(* Logix 5000 project; controller grafcet1 Emulate 5570 rev 32.11; software revision 32.00 *)

TASK MainTask (continuous, watchdog 500 ms) : MainProgram

MODULES
   Local : Emulate 5570 (ICP 2, rev 32.11)
END_MODULES

VAR_GLOBAL   (* controller tags *)
   AlarmaWrapDone : BOOL;
   Banda2ON : BOOL;
   Bandallenado : BOOL;
   BandaON : BOOL;
   BandaRechazo : BOOL;
   BandaSalida : BOOL;
   BandaTapado : BOOL;
   Cocacola6 : BOOL;
   ContadorSecuencia : DINT;
   ContadorSensorRechazo : DINT := 61;
   ContadorWrap : COUNTER := (PRE := 18, ACC := 1);
   Cortadora : BOOL;
   CrearCocacolaWrap : BOOL;
   E0 : BOOL;
   E1 : BOOL;
   E10 : BOOL;
   E11 : BOOL;
   E12 : BOOL;
   E13 : BOOL;
   E14 : BOOL;
   E15 : BOOL;
   E16 : BOOL;
   E17 : BOOL;
   E18 : BOOL;
   E19 : BOOL;
   E2 : BOOL;
   E20 : BOOL;
   E21 : BOOL;
   E22 : BOOL;
   E3 : BOOL;
   E4 : BOOL;
   E5 : BOOL;
   E6 : BOOL;
   E7 : BOOL;
   E8 : BOOL;
   E9 : BOOL;
   EliminarCocacola6 : BOOL;
   EliminarCocacolaWrap : BOOL;
   EmergencyStop : BOOL := 1;
   EN_Lineas : BOOL;
   ER2 : BOOL;
   FechaHora : DINT[7];
   GenerarCocacola6 : BOOL;
   HornoON : BOOL;
   InterceptorGiro : DINT;
   Llenador : BOOL;
   Memoria_ONS : BOOL;
   NuevaBotella : BOOL;
   NuevaBotella_Ant : BOOL;
   NumeroBotellas : COUNTER := (PRE := 1000);
   NumeroBotellasRechazadas : COUNTER := (PRE := 1000);
   NumeroLote : DINT;
   ObjetoEnHorno : BOOL;
   OffsetLote : DINT;
   ONS_Llenado : BOOL;
   ONS_SalidaTapado : BOOL;
   ONS_Secuencia : BOOL;
   PistonRechazo : BOOL;
   PorcentajeRechazo : DINT := 20;
   PosicionLote : DINT;
   PulsadorRechazo : BOOL;
   RechazoAleatorio : BOOL;
   RechazosPor10 : DINT;
   Reset : BOOL;
   Rodillos : BOOL;
   RutinaPaletizado : BOOL;
   SeisBotellasWrap : COUNTER := (PRE := 6);
   SensorCortador : BOOL;
   SensorEntraBandaSW : BOOL;
   SensorInterceptor : BOOL;
   SensorInterceptorTrabajo : BOOL;
   SensorLlenado : BOOL;
   SensorPosicionRechazo : BOOL;
   SensorPosicionRechazo_Ant : BOOL;
   SensorSaleTunelCalor : BOOL;
   SensorSalidaBandaSW : BOOL;
   SensorSalidaRechazo : BOOL;
   SensorSalidaTapado : BOOL;
   SensorTapado : BOOL;
   SensorTope : BOOL;
   SensorTunelCalor : BOOL;
   START : BOOL;
   StartCalidad : BOOL;
   StartLlenado : BOOL;
   Tapado : BOOL;
   TerminaMov : BOOL;
   TiempoWrap : TIMER := (PRE := 2000);
   Tope : BOOL;
   TuboAbajo : BOOL;
   ValorAleatorio : DINT;
END_VAR

PROGRAM MainProgram   (* main routine MainRoutine *)

ROUTINE MainRoutine   (* ladder *)
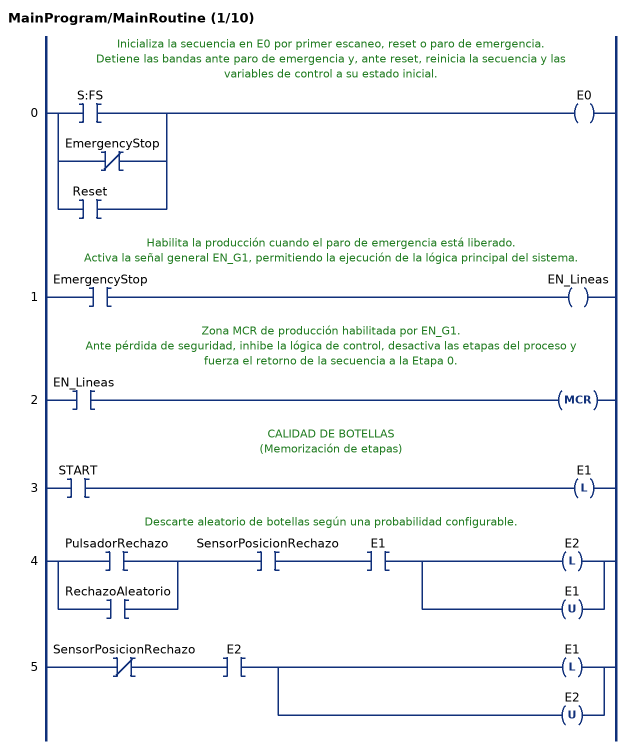
   // Inicializa la secuencia en E0 por primer escaneo, reset o paro de emergencia.
   // Detiene las bandas ante paro de emergencia y, ante reset, reinicia la secuencia y las variables de control a su estado inicial.
   0: [XIC(S:FS) ,XIO(EmergencyStop) ,XIC(Reset) ]OTE(E0);
   // Habilita la producción cuando el paro de emergencia está liberado.
   // Activa la señal general EN_G1, permitiendo la ejecución de la lógica principal del sistema.
   1: XIC(EmergencyStop)OTE(EN_Lineas);
   // Zona MCR de producción habilitada por EN_G1.
   // Ante pérdida de seguridad, inhibe la lógica de control, desactiva las etapas del proceso y fuerza el retorno de la secuencia a la Etapa 0.
   2: XIC(EN_Lineas)MCR();
   // CALIDAD DE BOTELLAS
   // (Memorización de etapas)
   3: XIC(START)OTL(E1);
   // Descarte aleatorio de botellas según una probabilidad configurable.
   4: [XIC(PulsadorRechazo) ,XIC(RechazoAleatorio) ]XIC(SensorPosicionRechazo)XIC(E1)[OTL(E2) ,OTU(E1) ];
   5: XIO(SensorPosicionRechazo)XIC(E2)[OTL(E1) ,OTU(E2) ];
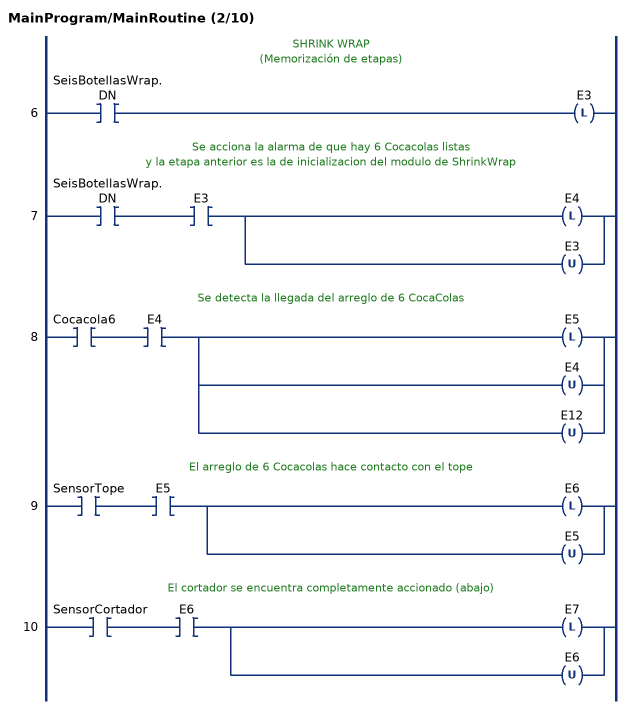
   // SHRINK WRAP
   //  (Memorización de etapas)
   6: XIC(SeisBotellasWrap.DN)OTL(E3);
   // Se acciona la alarma de que hay 6 Cocacolas listas
   // y la etapa anterior es la de inicializacion del modulo de ShrinkWrap
   7: XIC(SeisBotellasWrap.DN)XIC(E3)[OTL(E4) ,OTU(E3) ];
   // Se detecta la llegada del arreglo de 6 CocaColas
   8: XIC(Cocacola6)XIC(E4)[OTL(E5) ,OTU(E4) ,OTU(E12) ];
   // El arreglo de 6 Cocacolas hace contacto con el tope
   9: XIC(SensorTope)XIC(E5)[OTL(E6) ,OTU(E5) ];
   // El cortador se encuentra completamente accionado (abajo)
   10: XIC(SensorCortador)XIC(E6)[OTL(E7) ,OTU(E6) ];
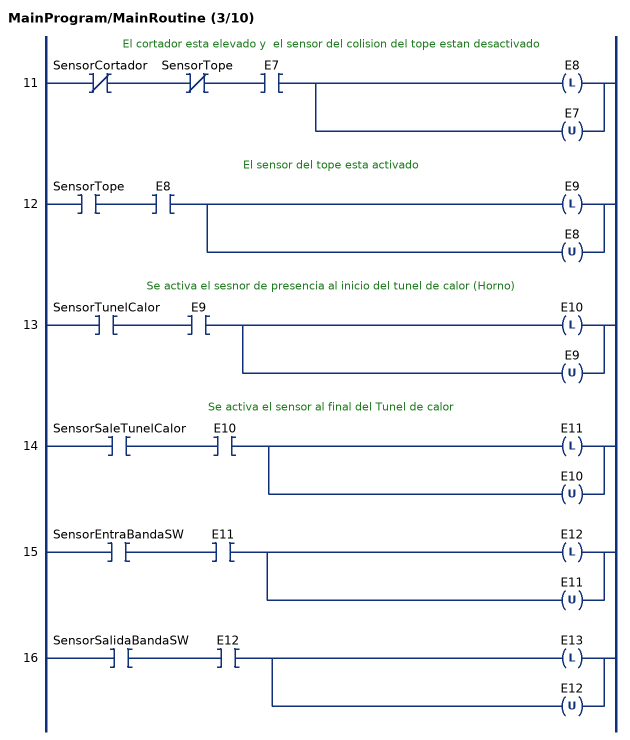
   // El cortador esta elevado y  el sensor del colision del tope estan desactivado
   11: XIO(SensorCortador)XIO(SensorTope)XIC(E7)[OTL(E8) ,OTU(E7) ];
   // El sensor del tope esta activado
   12: XIC(SensorTope)XIC(E8)[OTL(E9) ,OTU(E8) ];
   // Se activa el sesnor de presencia al inicio del tunel de calor (Horno)
   13: XIC(SensorTunelCalor)XIC(E9)[OTL(E10) ,OTU(E9) ];
   // Se activa el sensor al final del Tunel de calor
   14: XIC(SensorSaleTunelCalor)XIC(E10)[OTL(E11) ,OTU(E10) ];
   15: XIC(SensorEntraBandaSW)XIC(E11)[OTL(E12) ,OTU(E11) ];
   16: XIC(SensorSalidaBandaSW)XIC(E12)[OTL(E13) ,OTU(E12) ];
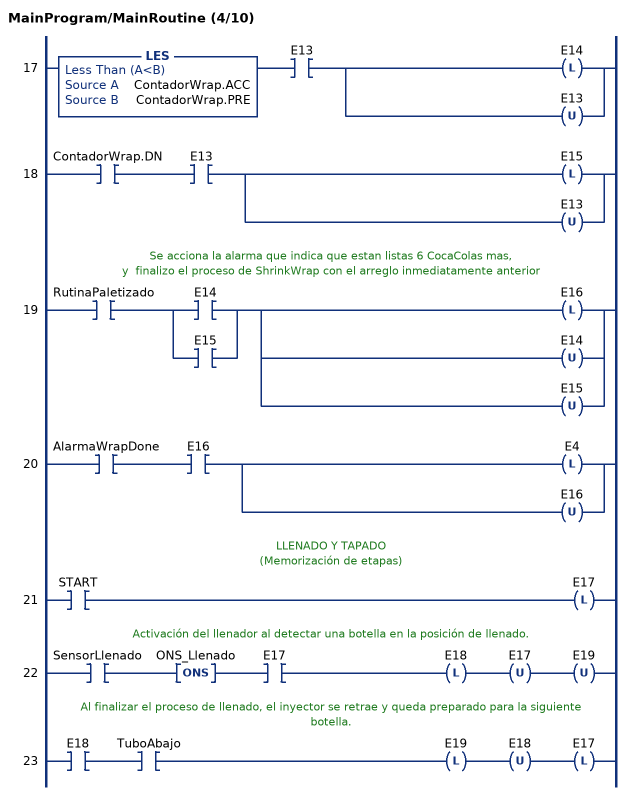
   17: LES(ContadorWrap.ACC,ContadorWrap.PRE)XIC(E13)[OTL(E14) ,OTU(E13) ];
   18: XIC(ContadorWrap.DN)XIC(E13)[OTL(E15) ,OTU(E13) ];
   // Se acciona la alarma que indica que estan listas 6 CocaColas mas,
   // y  finalizo el proceso de ShrinkWrap con el arreglo inmediatamente anterior
   19: XIC(RutinaPaletizado)[XIC(E14) ,XIC(E15) ][[OTL(E16) ,OTU(E14) ] ,OTU(E15) ];
   20: XIC(AlarmaWrapDone)XIC(E16)[OTL(E4) ,OTU(E16) ];
   // LLENADO Y TAPADO
   // (Memorización de etapas)
   21: XIC(START)OTL(E17);
   // Activación del llenador al detectar una botella en la posición de llenado.
   22: XIC(SensorLlenado)ONS(ONS_Llenado)XIC(E17)OTL(E18)OTU(E17)OTU(E19);
   // Al finalizar el proceso de llenado, el inyector se retrae y queda preparado para la siguiente botella.
   23: XIC(E18)XIC(TuboAbajo)OTL(E19)OTU(E18)OTL(E17);
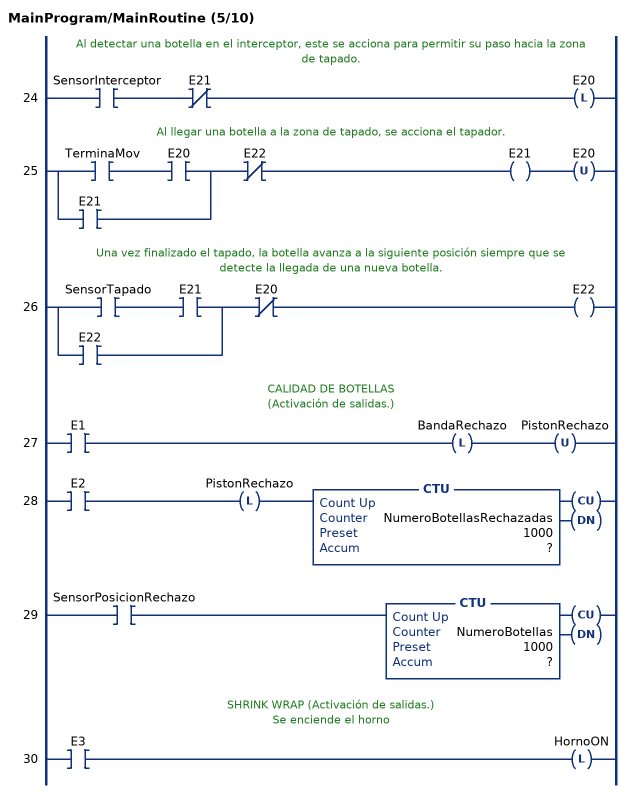
   // Al detectar una botella en el interceptor, este se acciona para permitir su paso hacia la zona de tapado.
   24: XIC(SensorInterceptor)XIO(E21)OTL(E20);
   // Al llegar una botella a la zona de tapado, se acciona el tapador.
   25: [XIC(TerminaMov) XIC(E20) ,XIC(E21) ]XIO(E22)OTE(E21)OTU(E20);
   // Una vez finalizado el tapado, la botella avanza a la siguiente posición siempre que se detecte la llegada de una nueva botella.
   26: [XIC(SensorTapado) XIC(E21) ,XIC(E22) ]XIO(E20)OTE(E22);
   // CALIDAD DE BOTELLAS
   // (Activación de salidas.)
   27: XIC(E1)OTL(BandaRechazo)OTU(PistonRechazo);
   28: XIC(E2)OTL(PistonRechazo)CTU(NumeroBotellasRechazadas,?,?);
   29: XIC(SensorPosicionRechazo)CTU(NumeroBotellas,?,?);
   // SHRINK WRAP (Activación de salidas.)
   // Se enciende el horno
   30: XIC(E3)OTL(HornoON);
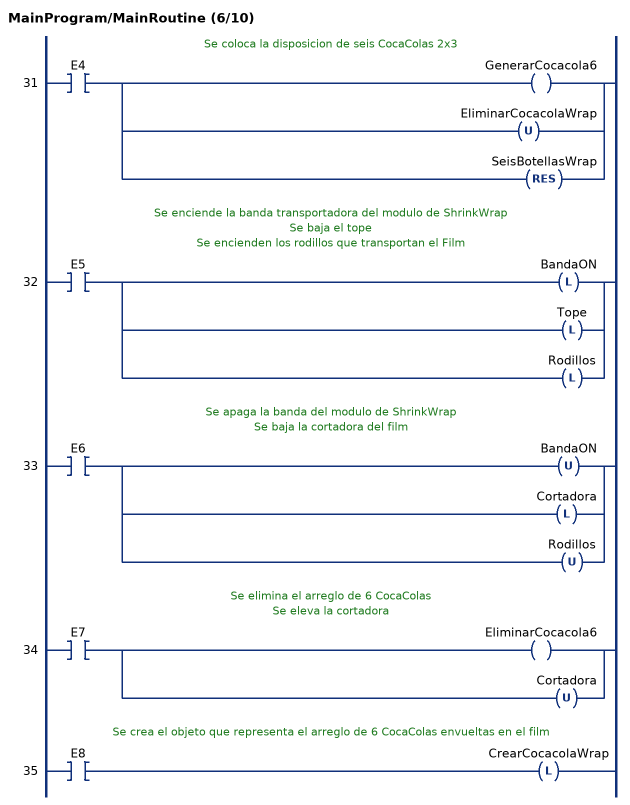
   // Se coloca la disposicion de seis CocaColas 2x3
   31: XIC(E4)[OTE(GenerarCocacola6) ,[OTU(EliminarCocacolaWrap) ,RES(SeisBotellasWrap) ] ];
   // Se enciende la banda transportadora del modulo de ShrinkWrap
   // Se baja el tope
   // Se encienden los rodillos que transportan el Film
   32: XIC(E5)[[OTL(BandaON) ,OTL(Tope) ] ,OTL(Rodillos) ];
   // Se apaga la banda del modulo de ShrinkWrap
   // Se baja la cortadora del film
   33: XIC(E6)[[OTU(BandaON) ,OTL(Cortadora) ] ,OTU(Rodillos) ];
   // Se elimina el arreglo de 6 CocaColas
   // Se eleva la cortadora
   34: XIC(E7)[OTE(EliminarCocacola6) ,OTU(Cortadora) ];
   // Se crea el objeto que representa el arreglo de 6 CocaColas envueltas en el film
   35: XIC(E8)OTL(CrearCocacolaWrap);
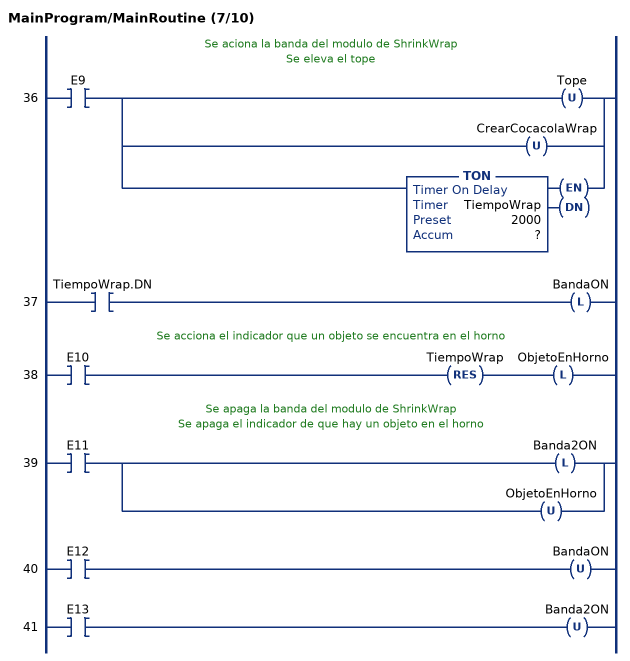
   // Se aciona la banda del modulo de ShrinkWrap
   // Se eleva el tope
   36: XIC(E9)[OTU(Tope) ,OTU(CrearCocacolaWrap) ,TON(TiempoWrap,?,?) ];
   37: XIC(TiempoWrap.DN)OTL(BandaON);
   // Se acciona el indicador que un objeto se encuentra en el horno
   38: XIC(E10)RES(TiempoWrap)OTL(ObjetoEnHorno);
   // Se apaga la banda del modulo de ShrinkWrap
   // Se apaga el indicador de que hay un objeto en el horno
   39: XIC(E11)[OTL(Banda2ON) ,OTU(ObjetoEnHorno) ];
   40: XIC(E12)OTU(BandaON);
   41: XIC(E13)OTU(Banda2ON);
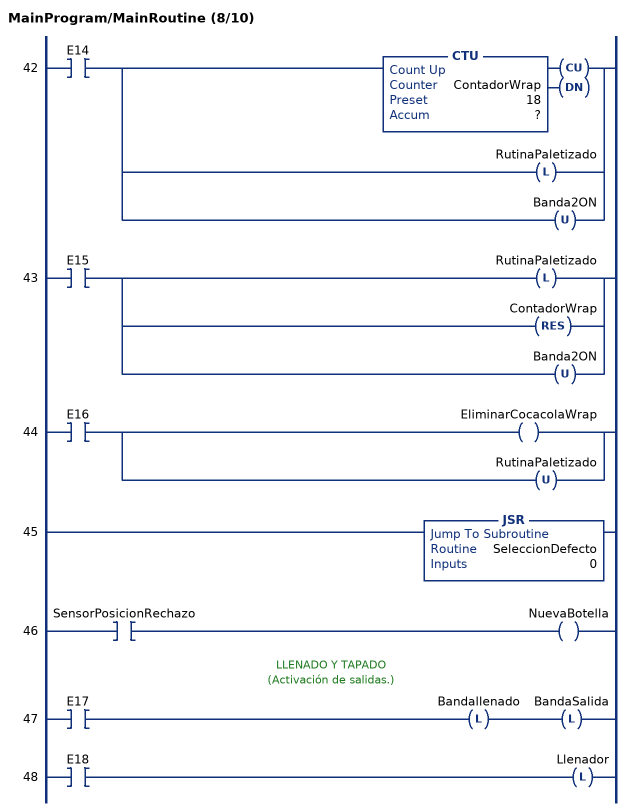
   42: XIC(E14)[[CTU(ContadorWrap,?,?) ,OTL(RutinaPaletizado) ] ,OTU(Banda2ON) ];
   43: XIC(E15)[[OTL(RutinaPaletizado) ,RES(ContadorWrap) ] ,OTU(Banda2ON) ];
   44: XIC(E16)[OTE(EliminarCocacolaWrap) ,OTU(RutinaPaletizado) ];
   45: JSR(SeleccionDefecto,0);
   46: XIC(SensorPosicionRechazo)OTE(NuevaBotella);
   // LLENADO Y TAPADO
   // (Activación de salidas.)
   47: XIC(E17)OTL(Bandallenado)OTL(BandaSalida);
   48: XIC(E18)OTL(Llenador);
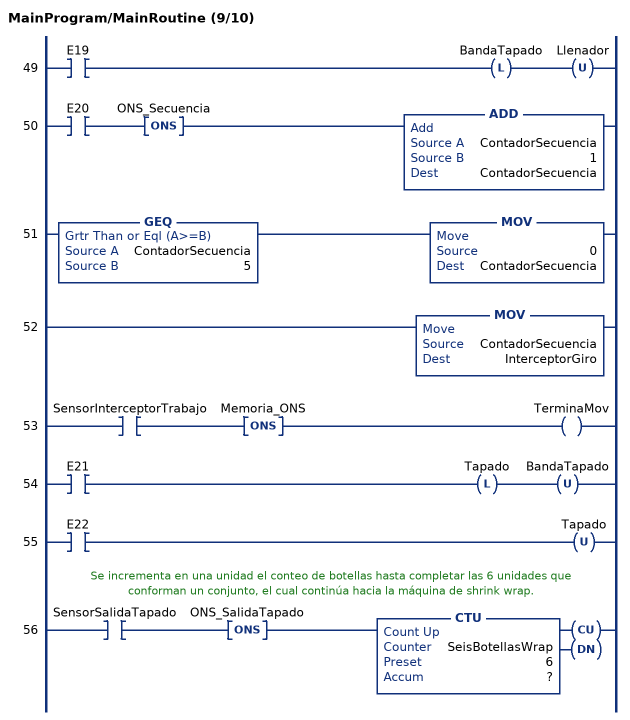
   49: XIC(E19)OTL(BandaTapado)OTU(Llenador);
   50: XIC(E20)ONS(ONS_Secuencia)ADD(ContadorSecuencia,1,ContadorSecuencia);
   51: GEQ(ContadorSecuencia,5)MOV(0,ContadorSecuencia);
   52: MOV(ContadorSecuencia,InterceptorGiro);
   53: XIC(SensorInterceptorTrabajo)ONS(Memoria_ONS)OTE(TerminaMov);
   54: XIC(E21)OTL(Tapado)OTU(BandaTapado);
   55: XIC(E22)OTU(Tapado);
   // Se incrementa en una unidad el conteo de botellas hasta completar las 6 unidades que conforman un conjunto, el cual continúa hacia la máquina de shrink wrap.
   56: XIC(SensorSalidaTapado)ONS(ONS_SalidaTapado)CTU(SeisBotellasWrap,?,?);
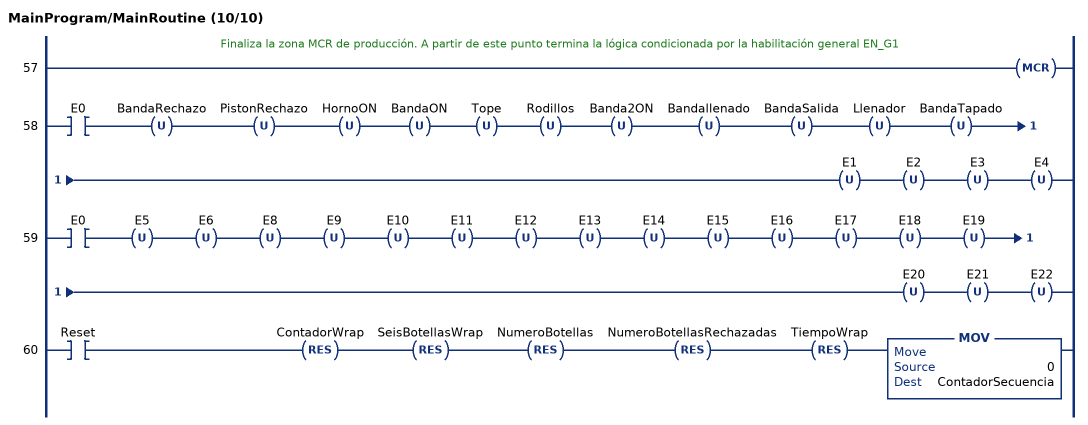
   // Finaliza la zona MCR de producción. A partir de este punto termina la lógica condicionada por la habilitación general EN_G1
   57: MCR();
   58: XIC(E0)OTU(BandaRechazo)OTU(PistonRechazo)OTU(HornoON)OTU(BandaON)OTU(Tope)OTU(Rodillos)OTU(Banda2ON)OTU(Bandallenado)OTU(BandaSalida)OTU(Llenador)OTU(BandaTapado)OTU(E1)OTU(E2)OTU(E3)OTU(E4);
   59: XIC(E0)OTU(E5)OTU(E6)OTU(E8)OTU(E9)OTU(E10)OTU(E11)OTU(E12)OTU(E13)OTU(E14)OTU(E15)OTU(E16)OTU(E17)OTU(E18)OTU(E19)OTU(E20)OTU(E21)OTU(E22);
   60: XIC(Reset)RES(ContadorWrap)RES(SeisBotellasWrap)RES(NumeroBotellas)RES(NumeroBotellasRechazadas)RES(TiempoWrap)MOV(0,ContadorSecuencia);
END_ROUTINE

ROUTINE SeleccionDefecto   (* structured text *)
   // Detectar únicamente el flanco ascendente del sensor,
   // es decir, contar una sola vez cada botella que llega.
   IF SensorPosicionRechazo AND NOT SensorPosicionRechazo_Ant THEN
   
       // Contar la botella actual
       ContadorSensorRechazo := ContadorSensorRechazo + 1;
   
   
       // Decidir si esta botella debe rechazarse.
       //
       // Con PorcentajeRechazo = 20:
       // se rechazan exactamente 2 de cada 10 botellas.
       //
       // Con PorcentajeRechazo = 50:
       // se rechazan exactamente 5 de cada 10 botellas.
       //
       // El orden cambia entre grupos para que no sean consecutivas.
   
       IF (((((ContadorSensorRechazo - 1) MOD 10) * 7)
           + (((ContadorSensorRechazo - 1) / 10) * 3)) MOD 10)
           < (PorcentajeRechazo / 10) THEN
   
           RechazoAleatorio := 1;
   
       ELSE
   
           RechazoAleatorio := 0;
   
       END_IF;
   
   END_IF;
   
   
   // Cuando el sensor se desactiva, apagar la decisión de rechazo
   IF NOT SensorPosicionRechazo THEN
       RechazoAleatorio := 0;
   END_IF;
   
   
   // Guardar el estado anterior del sensor
   SensorPosicionRechazo_Ant := SensorPosicionRechazo;
END_ROUTINE
END_PROGRAM
